SUBAPPLICATION Uebung_090a1_AX (* Beispiel für AX_MUX_2 *)
  (* Standard: 61499-2; Description: Copyright (c) 2023 Meisterschulen am Ostbahnhof This program and the accompanying materials are made available under the terms of the Eclipse Public License 2.0 which is available at https://www.eclipse.org/legal/epl-2.0/ SPDX-License-Identifier: EPL-2.0 *)
  (* Version 1.0, 2023-10-23, Franz Höpfinger, Meisterschulen am Ostbahnhof, initial API and implementation and/or initial documentation *)
  PACKAGE Uebungen;
  IMPORT logiBUS::io::DI::logiBUS_DI::Input_I1;
  IMPORT logiBUS::io::DI::logiBUS_DI::Input_I2;
  IMPORT logiBUS::io::DI::logiBUS_DI::Input_I4;
  IMPORT logiBUS::io::DQ::logiBUS_DO::Output_Q1;
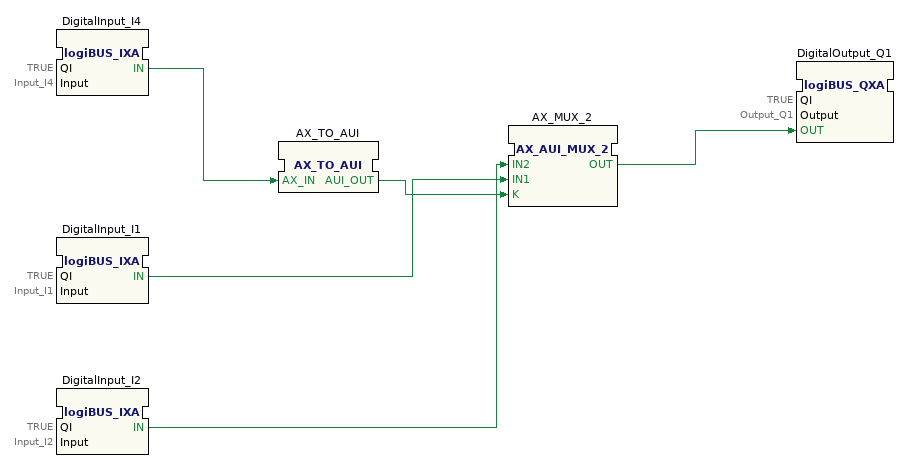
  FBS
    AX_MUX_2 : adapter::selection::unidirectional::AX_AUI_MUX_2;
    DigitalInput_I4 : logiBUS::io::DI::logiBUS_IXA(QI := TRUE, Input := Input_I4);
    DigitalOutput_Q1 : logiBUS::io::DQ::logiBUS_QXA(QI := TRUE, Output := Output_Q1);
    DigitalInput_I1 : logiBUS::io::DI::logiBUS_IXA(QI := TRUE, Input := Input_I1);
    DigitalInput_I2 : logiBUS::io::DI::logiBUS_IXA(QI := TRUE, Input := Input_I2);
    AX_TO_AUI : adapter::conversion::unidirectional::AX_TO_AUI;
  END_FBS
  ADAPTER_CONNECTIONS
    DigitalInput_I2.IN TO AX_MUX_2.IN2;
    DigitalInput_I1.IN TO AX_MUX_2.IN1;
    AX_MUX_2.OUT TO DigitalOutput_Q1.OUT;
    DigitalInput_I4.IN TO AX_TO_AUI.AX_IN;
    AX_TO_AUI.AUI_OUT TO AX_MUX_2.K;
  END_CONNECTIONS
END_SUBAPPLICATION
